ADAPTER EVENT_HS_UNI (* Handshake family, unidirectional fire-and-forget (dataless): REQ only, no reply *)
  (* Standard: 61499-1; Description: Copyright (c) 2026 HR Agrartechnik GmbH This program and the accompanying materials are made available under the terms of the Eclipse Public License 2.0 which is available at https://www.eclipse.org/legal/epl-2.0/ SPDX-License-Identifier: EPL-2.0 *)
  (* Version 1.0, 2026-09-02, Franz Höpfinger, HR Agrartechnik GmbH, Unidirectional, dataless reduction of EVENT_HS: only REQ, no CNF/IND/RSP at all - a pure fire-and-forget notification, not a real handshake (no acknowledgement, no way to know the Socket side received it) *)
  PACKAGE adapter::types::bidirectional::Handshake;
  (* Documentation:
  Reduced, unidirectional member of the EVENT_HS family (Handshake design pattern, IEC 61499 primer course, Module 6, Valeriy Vyatkin). Declares only a single REQ event, from Plug to Socket - no CNF, IND, or RSP at all.
   This is deliberately not a real handshake: the Socket side has no way to acknowledge or refuse the request, and the Plug side has no way to know whether the Socket ever received or reacted to it. Use this only for genuine fire-and-forget notifications where that one-way, best-effort semantics is actually acceptable - not as a drop-in replacement for EVENT_HS.
   Same Socket/Plug role split as EVENT_HS: Plug (Name>>) keeps the declared direction and fires REQ; Socket (>>Name) mirrors it and reacts to REQ.
   See test_AX/Meins/DesingPatterns/HandshakePattern/HandshakePattern.md for the full write-up of the EVENT_HS family, including this and the other three reduced variants (EVENT_HS_UNI_WSTRING, EVENT_HS_ACK, EVENT_HS_ACK_WSTRING).
  *)
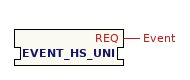
  EVENT_OUTPUT
    REQ; (* Request/notification from Plug to Socket, no reply expected *)
  END_EVENT
END_ADAPTER
